FUNCTION_BLOCK MockEventHandler IMPLEMENTS I_EventHandler
VAR
	_eventsHandled : INT;
	lastEventHandled : I_Event;
END_VAR

METHOD PUBLIC EqualsLastEvent : bool
VAR_INPUT
	Event : I_Event;
END_VAR
EqualsLastEvent := lastEventHandled = Event;
END_METHOD

PROPERTY EventsHandled : int
GET
EventsHandled := _eventsHandled;
END_GET
END_PROPERTY

METHOD HandleEvent
VAR_INPUT
	Event	: I_Event;
END_VAR
_eventsHandled := _eventsHandled + 1;
lastEventHandled := Event;
END_METHOD

END_FUNCTION_BLOCK

(* stored: Version 1.1.0.1, ProductVersion 3.1.4024.12
   POU MockEventHandler: Id {e5c40a76-6be0-0e8c-0e05-686c087ef0ee}, SpecialFunc None
   Method EqualsLastEvent: Id {571368ef-4b3a-012d-1567-fbfa76757fe9}
   Property EventsHandled: Id {42cd2462-2608-0be5-029b-b79da3772aeb}
   Get Get: Id {e57a048e-861f-057f-3abe-0f111a61f346}
   Method HandleEvent: Id {deed9fc6-275c-0842-21ab-1ab8f27699a5} *)
